(* PLC project Blank Project, Blank Blank 1.0 *)
(* stored: creationDateTime 2016-05-18T21:14:07, modificationDateTime 2019-07-16T18:46:01 *)

PROGRAM My_Program
  VAR
    button AT %IX0.0 : BOOL;
    sensor AT %IX0.1 : BOOL;
    lamp AT %QX0.0 : BOOL;
    switch AT %QX0.1 : BOOL;
  END_VAR
  VAR_INPUT
    test : BOOL;
  END_VAR
  VAR_OUTPUT
    test0 : BOOL;
  END_VAR
  VAR_IN_OUT
    test1 : BOOL;
  END_VAR
  VAR_EXTERNAL
    test2 : BOOL;
  END_VAR
  VAR_TEMP
    test3 : BOOL;
  END_VAR
  VAR
    T0 : TOF;
  END_VAR

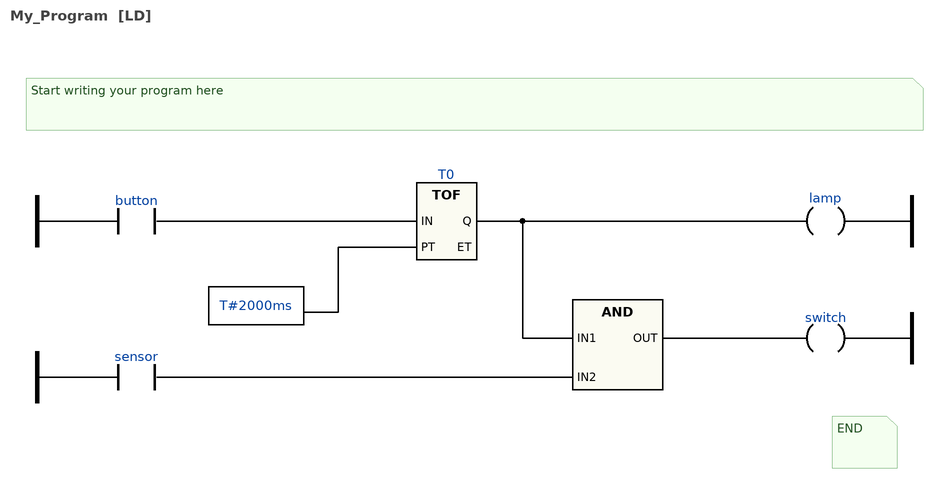
(* LD diagram, written out as Structured Text *)
(* Start writing your program here *)
T0(IN := button, PT := T#2000ms);
lamp := T0.Q;
switch := T0.Q AND sensor;
(* END *)
END_PROGRAM
